Staubli VAL3: VelocityCfg.pjx

--- VelocityCfg.pjx ---
Parameters version=s7.8.1 stackSize=5000 millimeterUnit=true
Program file=start.pgx
Program file=stop.pgx
Data file=VelocityCfg.dtx

--- VelocityCfg.dtx ---
public num nCmdType
public num nRefFrameVec[6]
public num nToolVec[6]
public num nAccel
public num nVel
public num nTransVel
public num nRotVel
